Staubli VAL3: loadmaster7.pgx

program loadmaster7(string x_sMasterFile7 (dimensions=1))
begin
  if master:libLoad(x_sMasterFile7)<0
    popUpMsg("nO ok")
  endIf
  frmaster[7].trsf=master:tTool.trsf
  //取个数
  nsize[7]=size(master:ptRoutingPath)
  //存个数
  resize(pdemo7,1,nsize[7])
  //保存程序
  master:libSave()
end
